// SIMATIC S7-200 SMART project (STEP 7-Micro/WIN SMART), CPU ST30

SYMBOL_TABLE 系统符号
Always_On        SM0.0    // 始终接通
First_Scan_On    SM0.1    // 仅在第一个扫描周期时接通
Time_0_Intrvl    SMB34    // 指定中断 0 的时间间隔（从 5 到 255，以 1 毫秒递增）。
END_SYMBOL_TABLE

ORGANIZATION_BLOCK MAIN:OB1
TITLE=程序注释
BEGIN
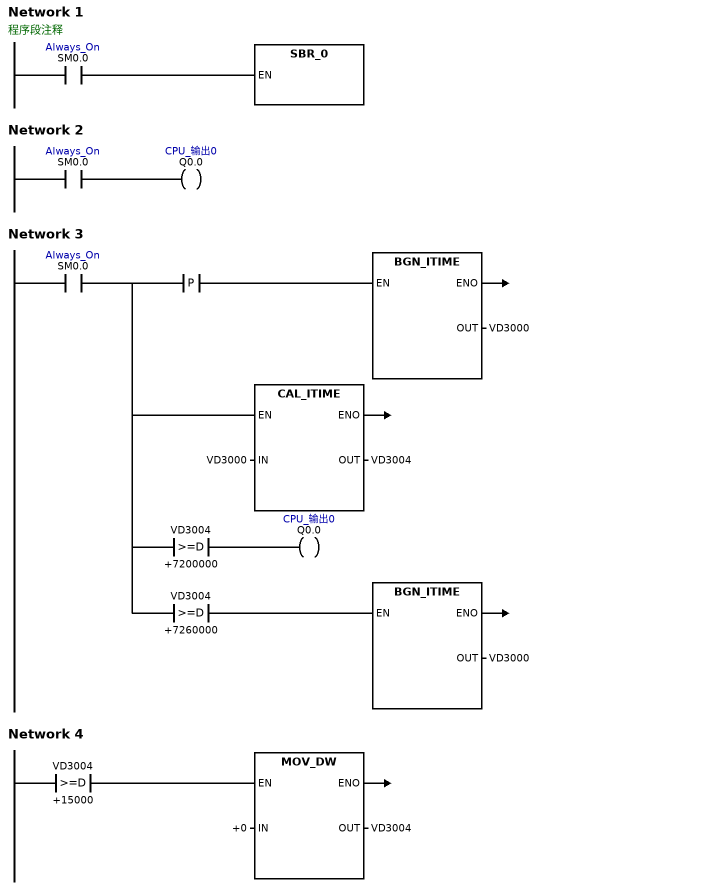
Network 1
// 程序段注释
LD     Always_On:SM0.0
CALL   SBR_0:SBR0
Network 2
LD     Always_On:SM0.0
=      CPU_输出0:Q0.0
Network 3
LD     Always_On:SM0.0
LPS
EU
BITIM  VD3000
LRD
CITIM  VD3000, VD3004
LRD
AD>=   VD3004, +7200000
=      CPU_输出0:Q0.0
LPP
AD>=   VD3004, +7260000
BITIM  VD3000
Network 4
LDD>=  VD3004, +15000
MOVD   +0, VD3004
END_ORGANIZATION_BLOCK

SUBROUTINE_BLOCK SBR_0:SBR0
TITLE=子程序注释
BEGIN
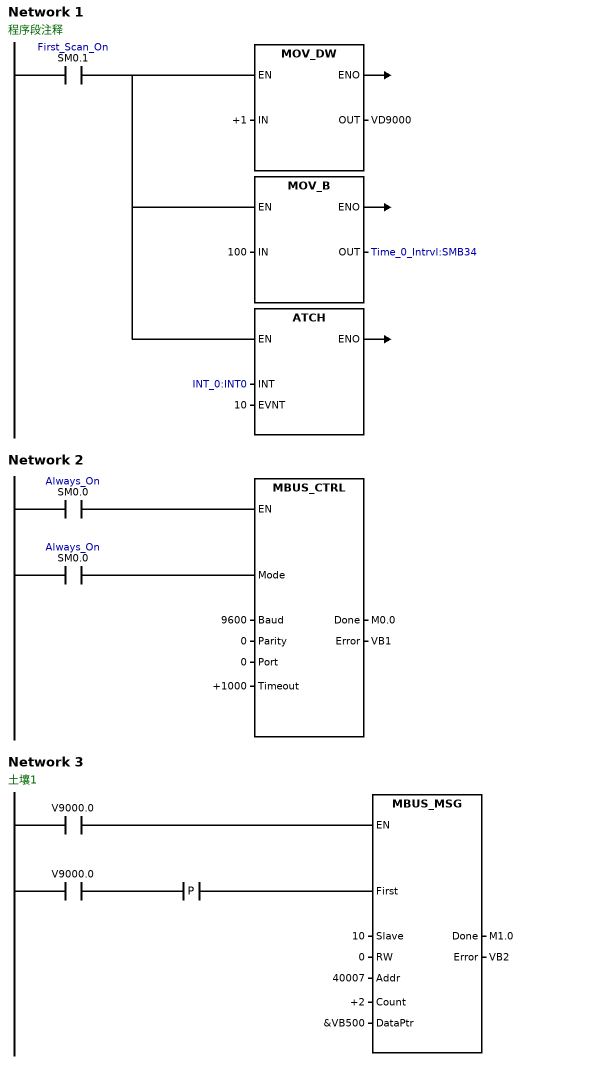
Network 1
// 程序段注释
LD     First_Scan_On:SM0.1
MOVD   +1, VD9000
MOVB   100, Time_0_Intrvl:SMB34
ATCH   INT_0:INT0, 10
Network 2
LD     Always_On:SM0.0
=      L60.0
LD     Always_On:SM0.0
=      L63.7
LD     L60.0
CALL   MBUS_CTRL:SBR1, L63.7, 9600, 0, 0, +1000, M0.0, VB1
Network 3
// 土壤1
LD     V9000.0
=      L60.0
LD     V9000.0
EU
=      L63.7
LD     L60.0
CALL   MBUS_MSG:SBR2, L63.7, 10, 0, 40007, +2, &VB500, M1.0, VB2
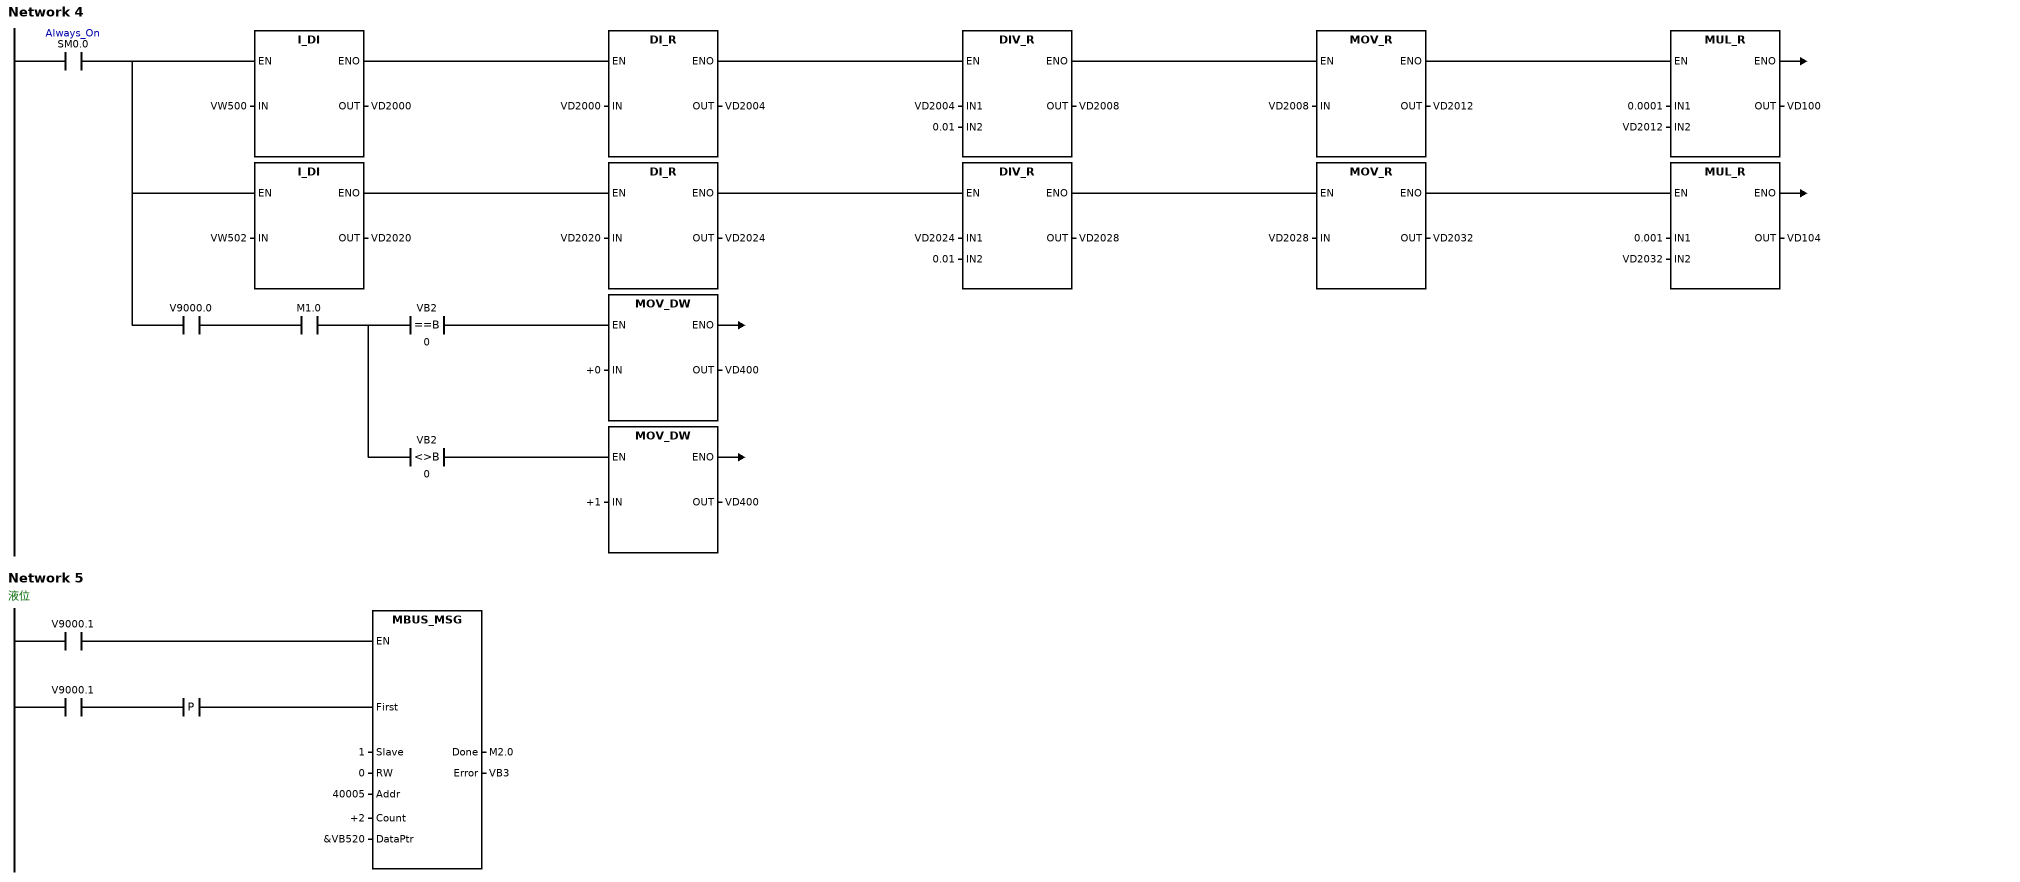
Network 4
LD     Always_On:SM0.0
LPS
ITD    VW500, VD2000
AENO
DTR    VD2000, VD2004
AENO
MOVR   VD2004, VD2008
AENO
/R     0.01, VD2008
AENO
MOVR   VD2008, VD2012
AENO
MOVR   0.0001, VD100
*R     VD2012, VD100
LRD
ITD    VW502, VD2020
AENO
DTR    VD2020, VD2024
AENO
MOVR   VD2024, VD2028
AENO
/R     0.01, VD2028
AENO
MOVR   VD2028, VD2032
AENO
MOVR   0.001, VD104
*R     VD2032, VD104
LPP
A      V9000.0
A      M1.0
LPS
AB=    VB2, 0
MOVD   +0, VD400
LPP
AB<>   VB2, 0
MOVD   +1, VD400
Network 5
// 液位
LD     V9000.1
=      L60.0
LD     V9000.1
EU
=      L63.7
LD     L60.0
CALL   MBUS_MSG:SBR2, L63.7, 1, 0, 40005, +2, &VB520, M2.0, VB3
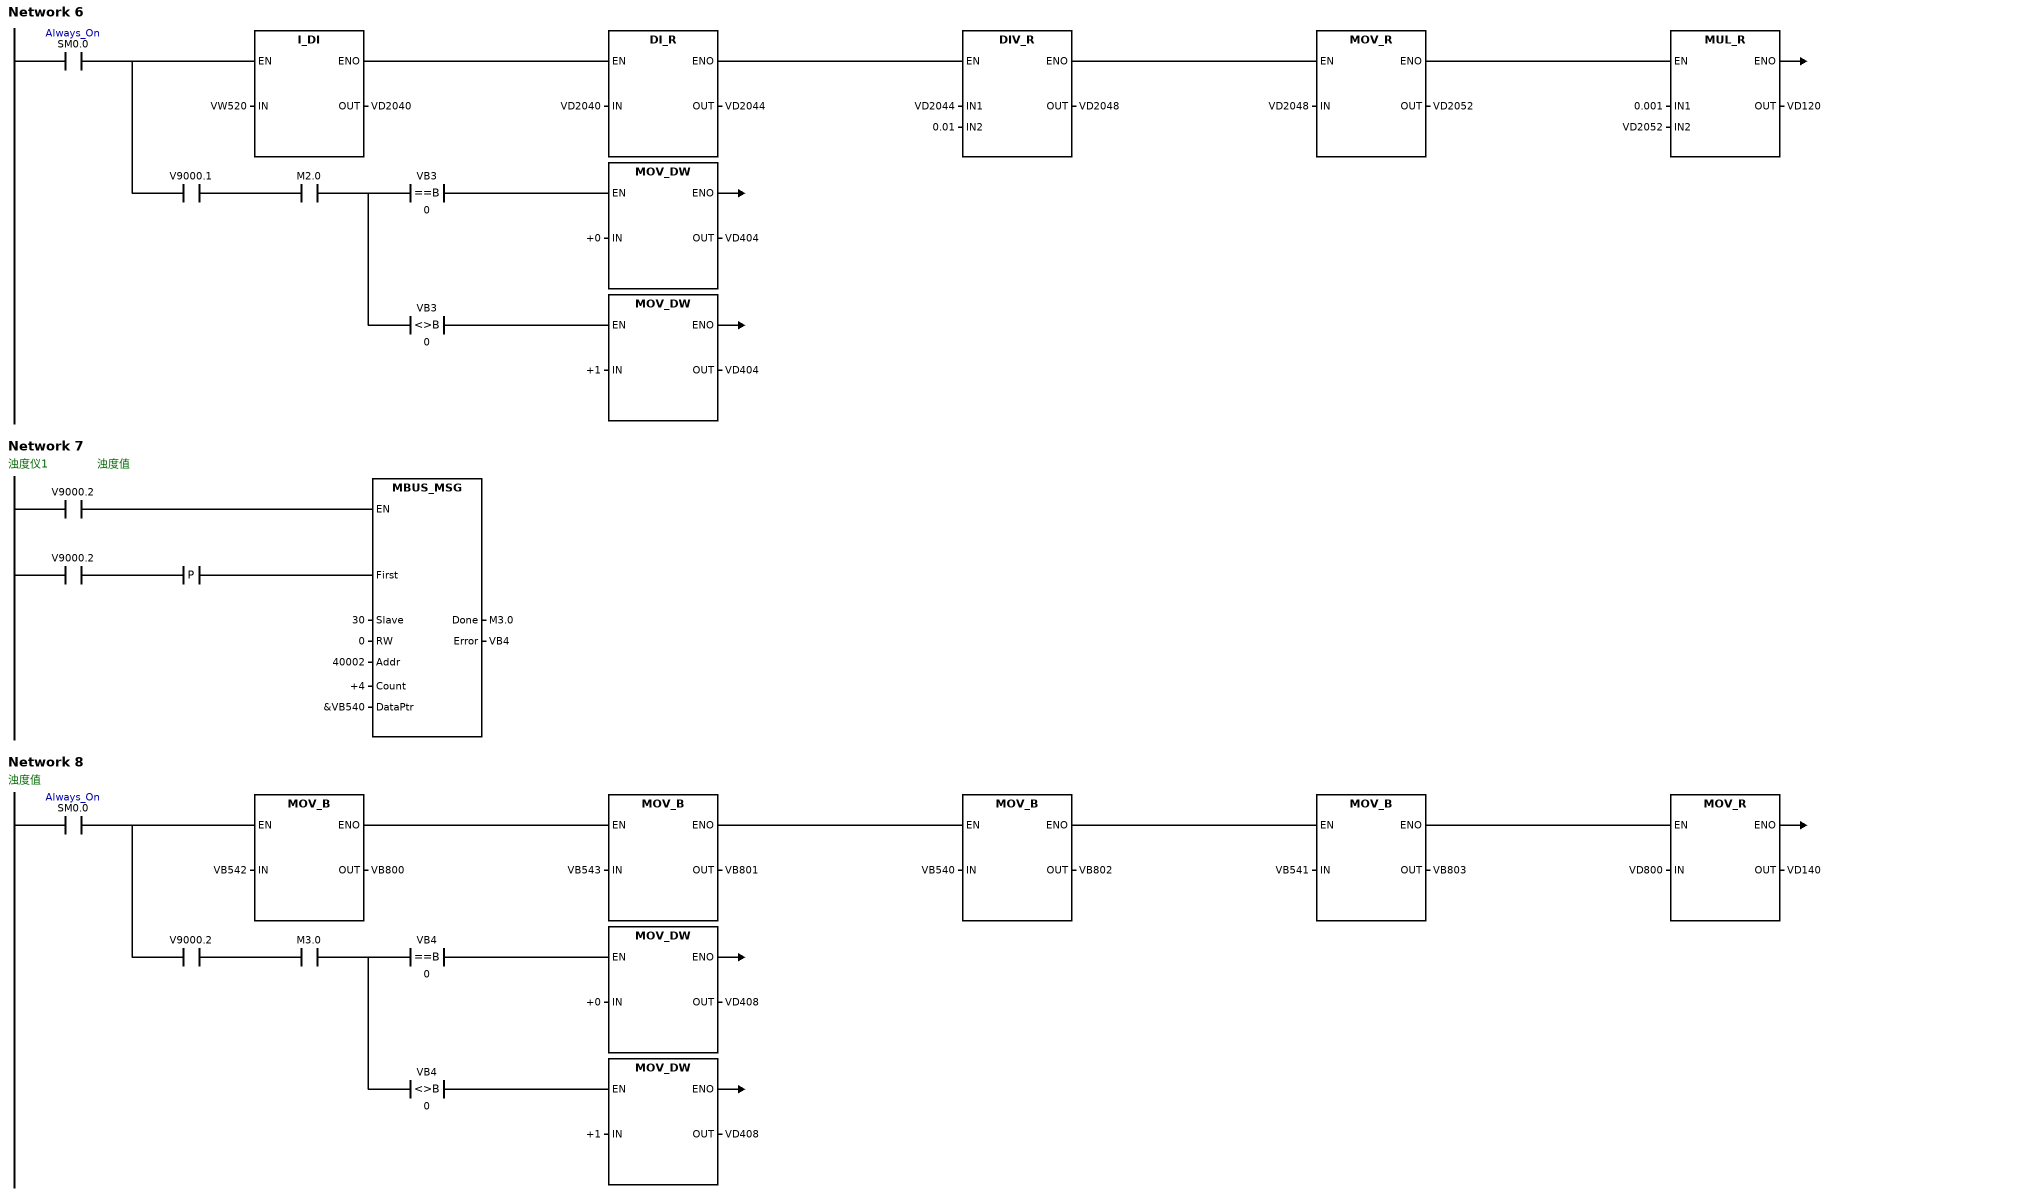
Network 6
LD     Always_On:SM0.0
LPS
ITD    VW520, VD2040
AENO
DTR    VD2040, VD2044
AENO
MOVR   VD2044, VD2048
AENO
/R     0.01, VD2048
AENO
MOVR   VD2048, VD2052
AENO
MOVR   0.001, VD120
*R     VD2052, VD120
LPP
A      V9000.1
A      M2.0
LPS
AB=    VB3, 0
MOVD   +0, VD404
LPP
AB<>   VB3, 0
MOVD   +1, VD404
Network 7
// 浊度仪1              浊度值
LD     V9000.2
=      L60.0
LD     V9000.2
EU
=      L63.7
LD     L60.0
CALL   MBUS_MSG:SBR2, L63.7, 30, 0, 40002, +4, &VB540, M3.0, VB4
Network 8
//  浊度值
LD     Always_On:SM0.0
LPS
MOVB   VB542, VB800
AENO
MOVB   VB543, VB801
AENO
MOVB   VB540, VB802
AENO
MOVB   VB541, VB803
AENO
MOVR   VD800, VD140
LPP
A      V9000.2
A      M3.0
LPS
AB=    VB4, 0
MOVD   +0, VD408
LPP
AB<>   VB4, 0
MOVD   +1, VD408
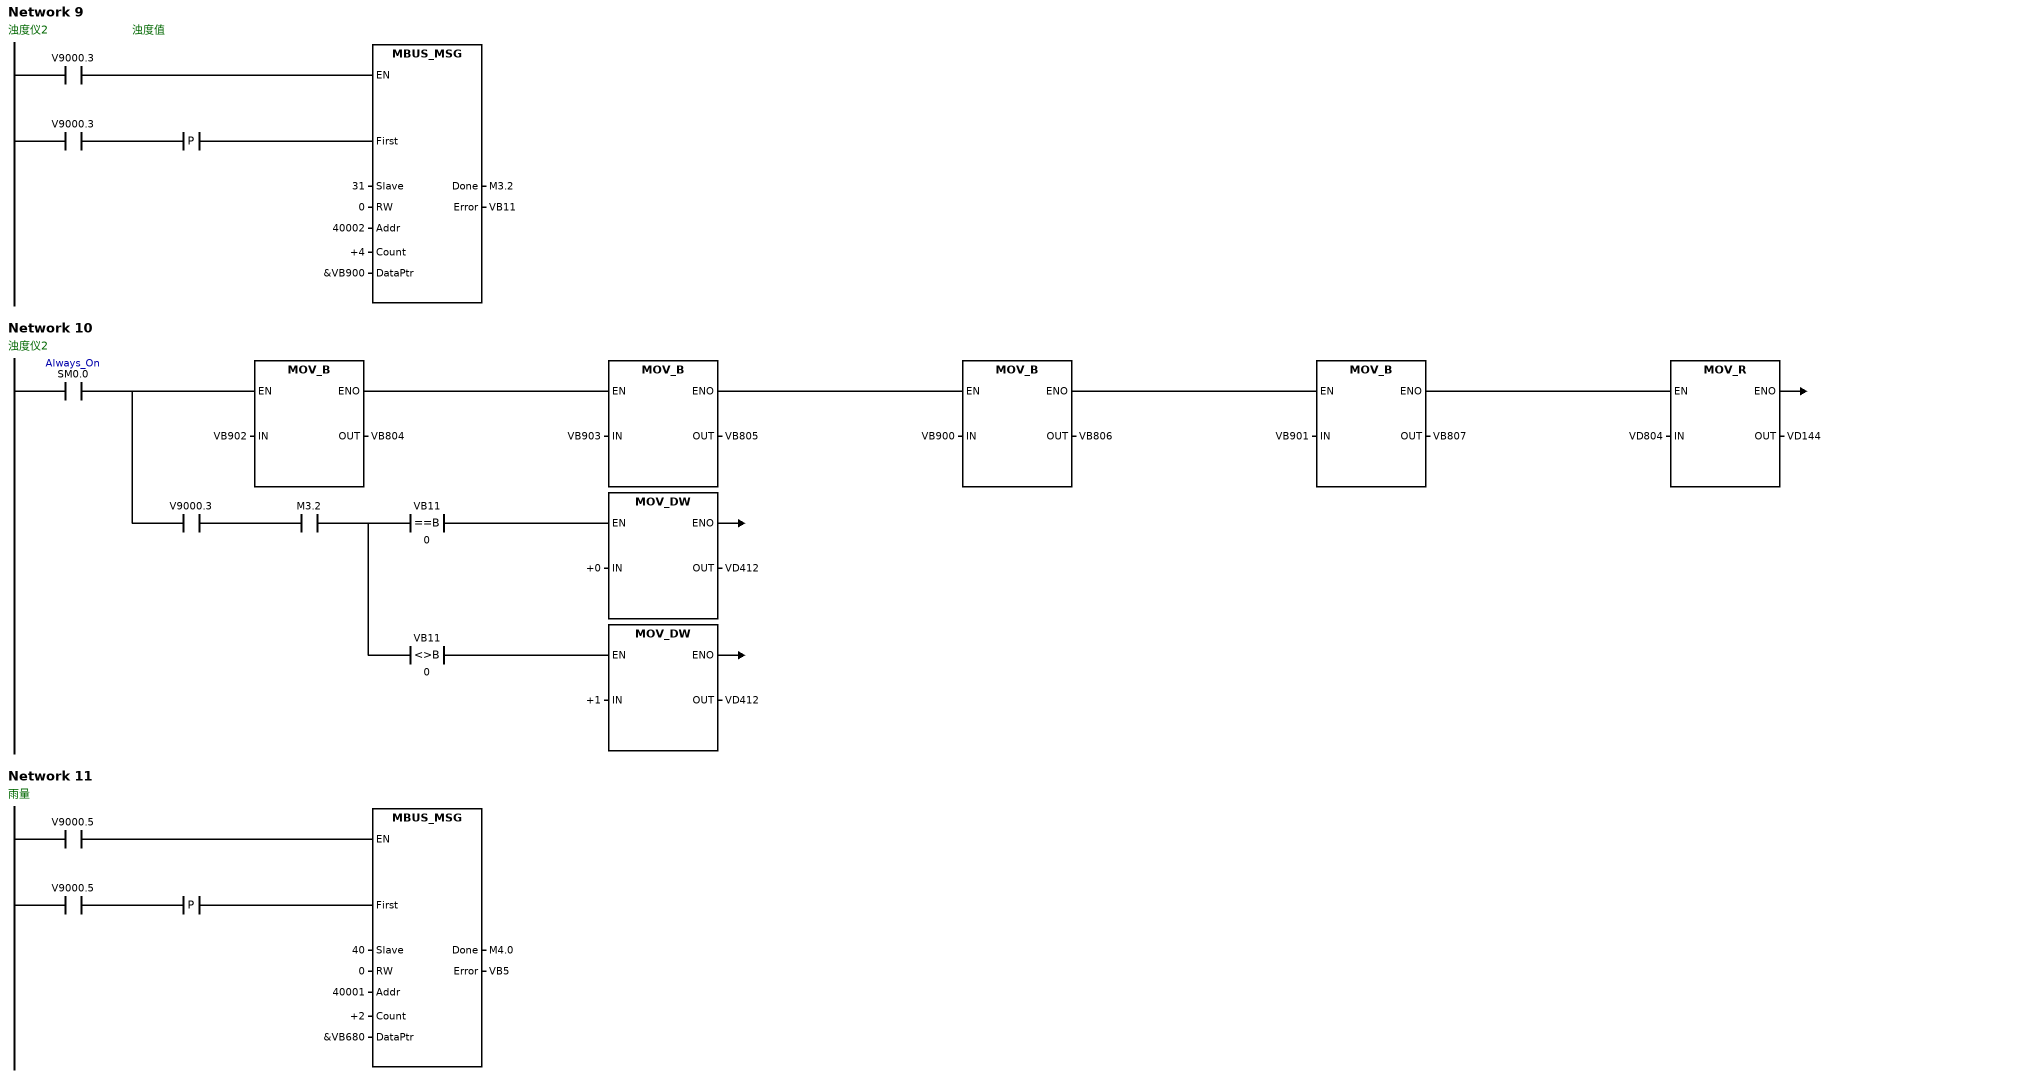
Network 9
// 浊度仪2                        浊度值
LD     V9000.3
=      L60.0
LD     V9000.3
EU
=      L63.7
LD     L60.0
CALL   MBUS_MSG:SBR2, L63.7, 31, 0, 40002, +4, &VB900, M3.2, VB11
Network 10
// 浊度仪2
LD     Always_On:SM0.0
LPS
MOVB   VB902, VB804
AENO
MOVB   VB903, VB805
AENO
MOVB   VB900, VB806
AENO
MOVB   VB901, VB807
AENO
MOVR   VD804, VD144
LPP
A      V9000.3
A      M3.2
LPS
AB=    VB11, 0
MOVD   +0, VD412
LPP
AB<>   VB11, 0
MOVD   +1, VD412
Network 11
// 雨量
LD     V9000.5
=      L60.0
LD     V9000.5
EU
=      L63.7
LD     L60.0
CALL   MBUS_MSG:SBR2, L63.7, 40, 0, 40001, +2, &VB680, M4.0, VB5
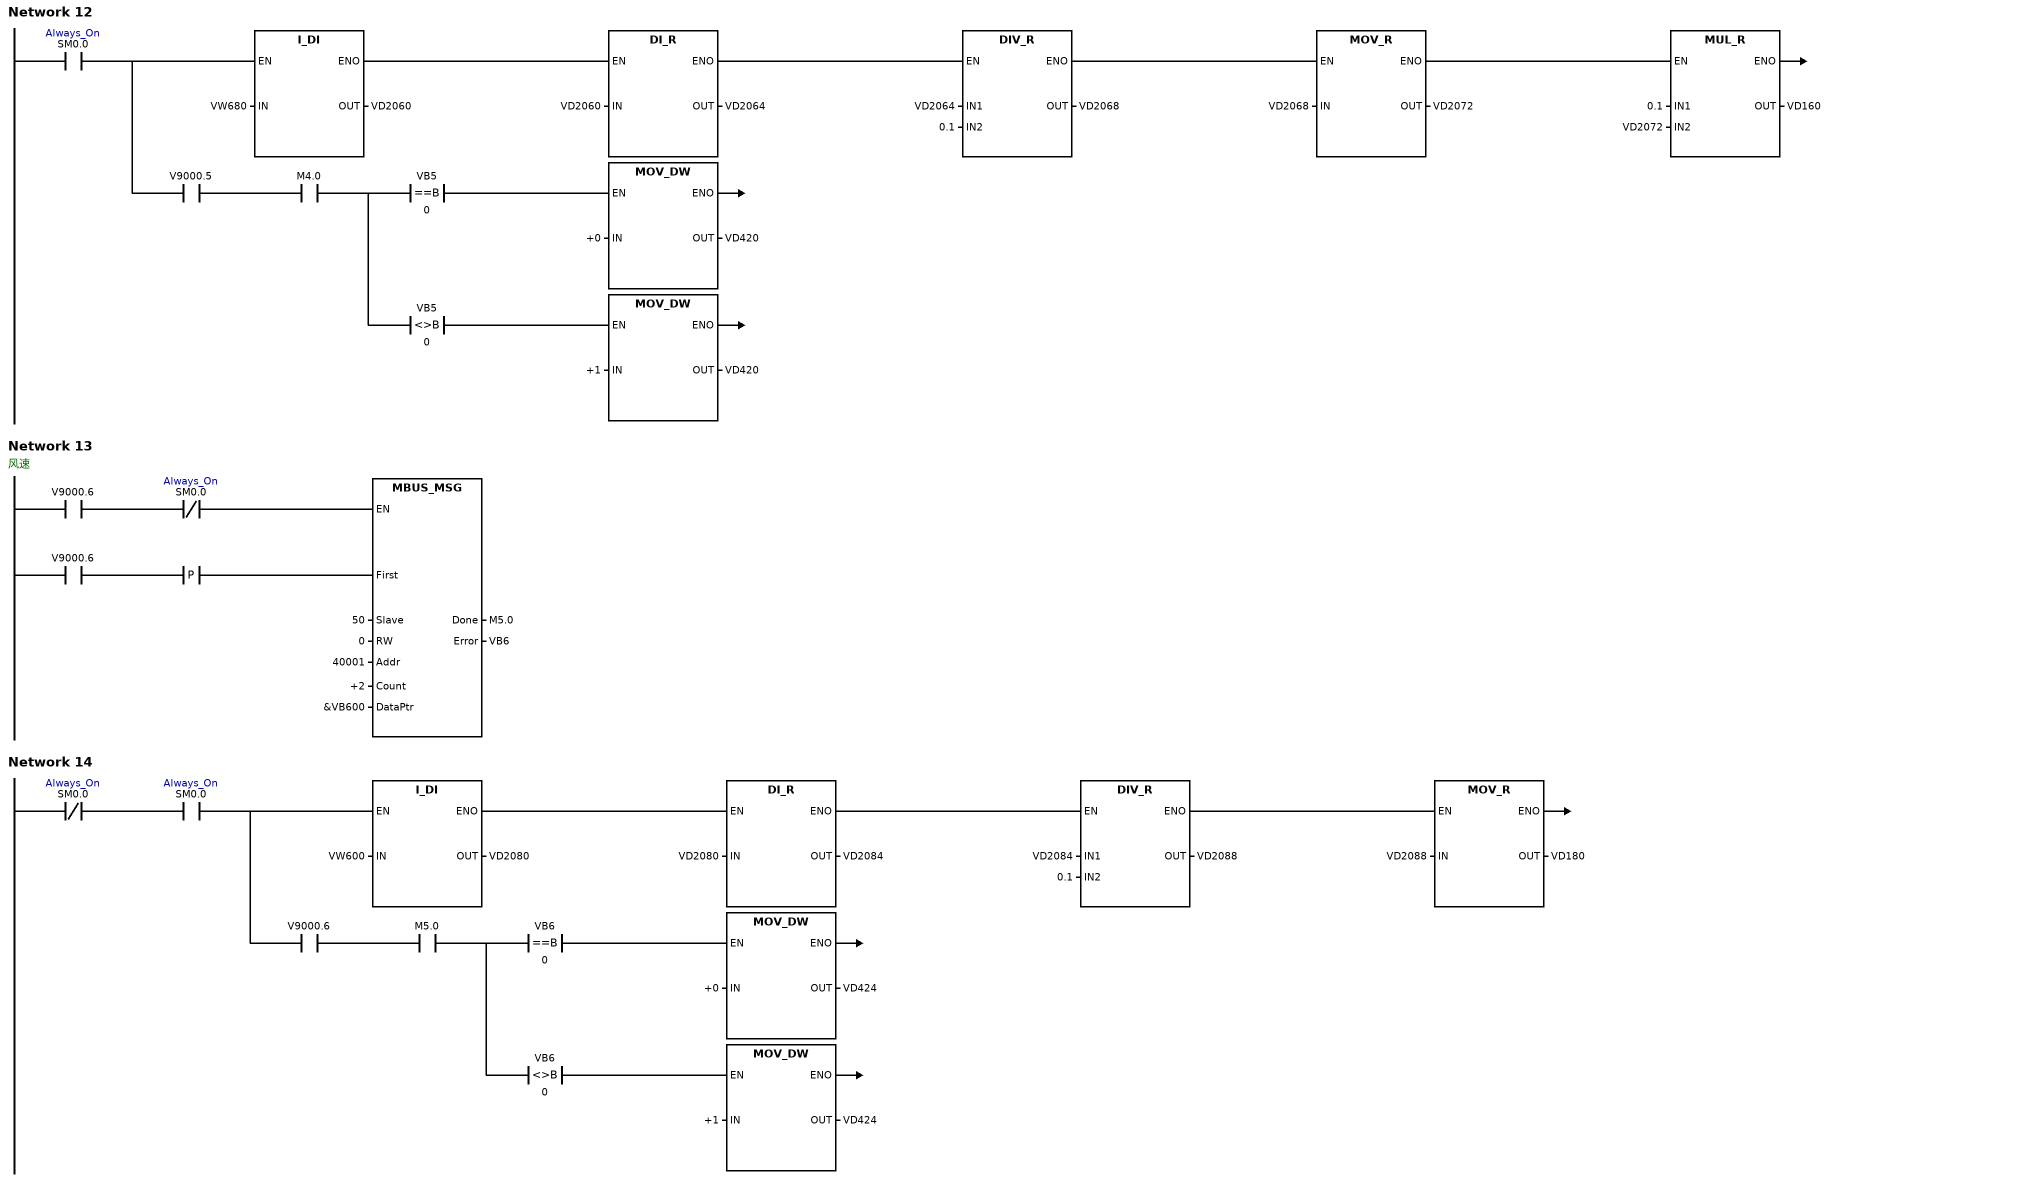
Network 12
LD     Always_On:SM0.0
LPS
ITD    VW680, VD2060
AENO
DTR    VD2060, VD2064
AENO
MOVR   VD2064, VD2068
AENO
/R     0.1, VD2068
AENO
MOVR   VD2068, VD2072
AENO
MOVR   0.1, VD160
*R     VD2072, VD160
LPP
A      V9000.5
A      M4.0
LPS
AB=    VB5, 0
MOVD   +0, VD420
LPP
AB<>   VB5, 0
MOVD   +1, VD420
Network 13
// 风速
LD     V9000.6
AN     Always_On:SM0.0
=      L60.0
LD     V9000.6
EU
=      L63.7
LD     L60.0
CALL   MBUS_MSG:SBR2, L63.7, 50, 0, 40001, +2, &VB600, M5.0, VB6
Network 14
LDN    Always_On:SM0.0
A      Always_On:SM0.0
LPS
ITD    VW600, VD2080
AENO
DTR    VD2080, VD2084
AENO
MOVR   VD2084, VD2088
AENO
/R     0.1, VD2088
AENO
MOVR   VD2088, VD180
LPP
A      V9000.6
A      M5.0
LPS
AB=    VB6, 0
MOVD   +0, VD424
LPP
AB<>   VB6, 0
MOVD   +1, VD424
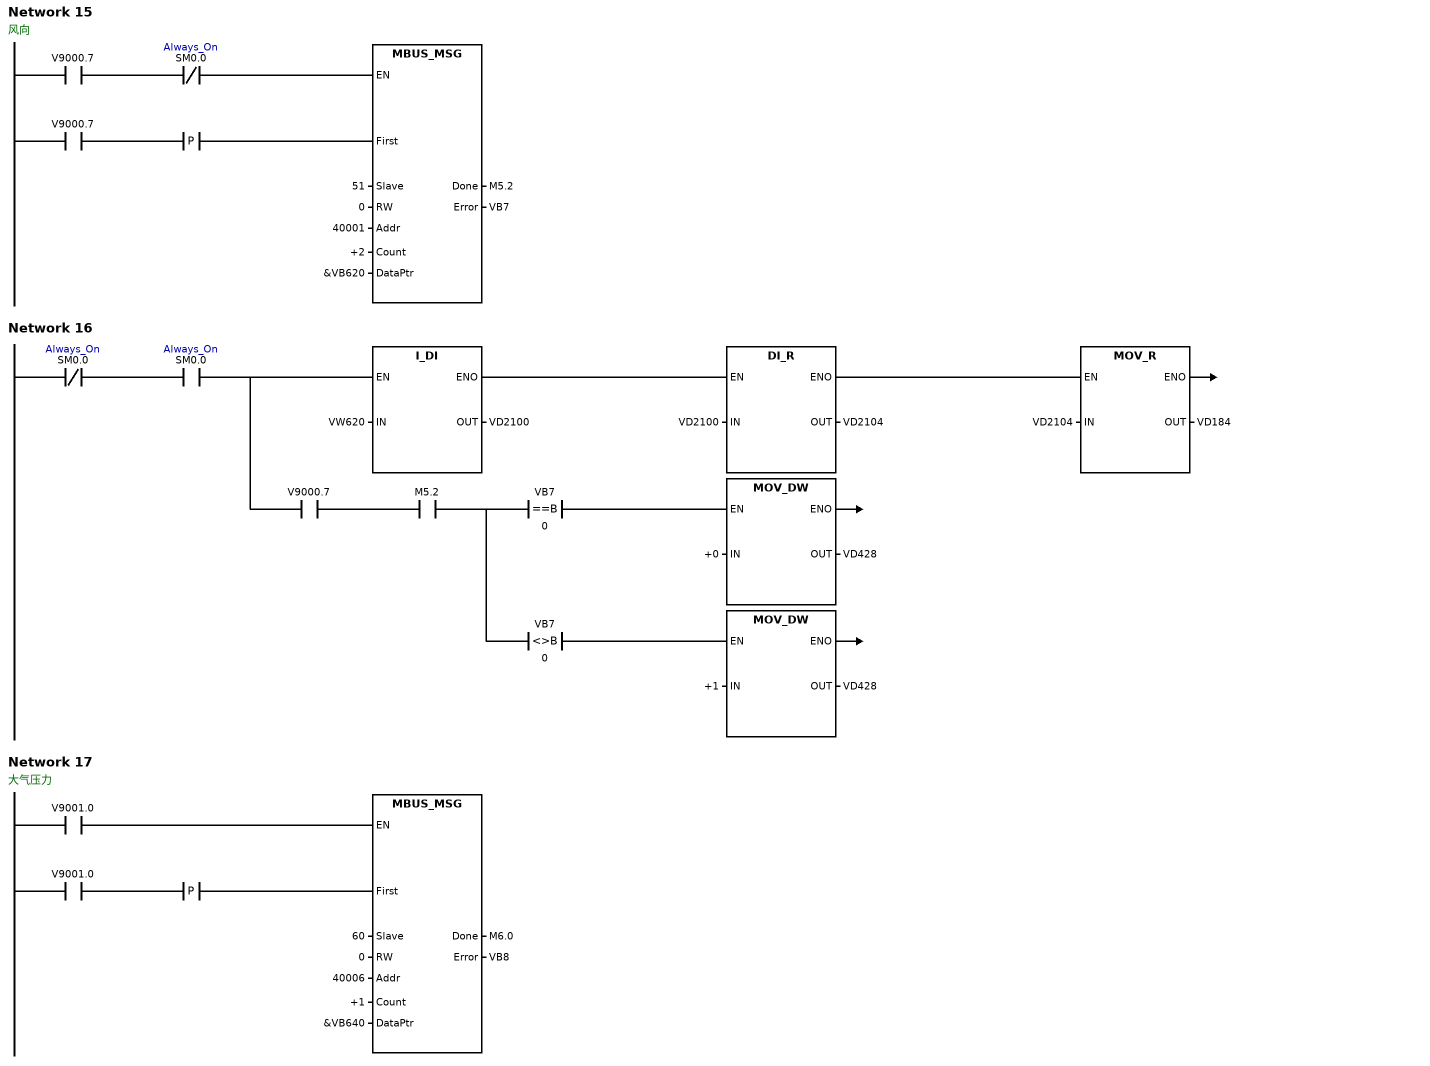
Network 15
// 风向
LD     V9000.7
AN     Always_On:SM0.0
=      L60.0
LD     V9000.7
EU
=      L63.7
LD     L60.0
CALL   MBUS_MSG:SBR2, L63.7, 51, 0, 40001, +2, &VB620, M5.2, VB7
Network 16
LDN    Always_On:SM0.0
A      Always_On:SM0.0
LPS
ITD    VW620, VD2100
AENO
DTR    VD2100, VD2104
AENO
MOVR   VD2104, VD184
LPP
A      V9000.7
A      M5.2
LPS
AB=    VB7, 0
MOVD   +0, VD428
LPP
AB<>   VB7, 0
MOVD   +1, VD428
Network 17
// 大气压力
LD     V9001.0
=      L60.0
LD     V9001.0
EU
=      L63.7
LD     L60.0
CALL   MBUS_MSG:SBR2, L63.7, 60, 0, 40006, +1, &VB640, M6.0, VB8
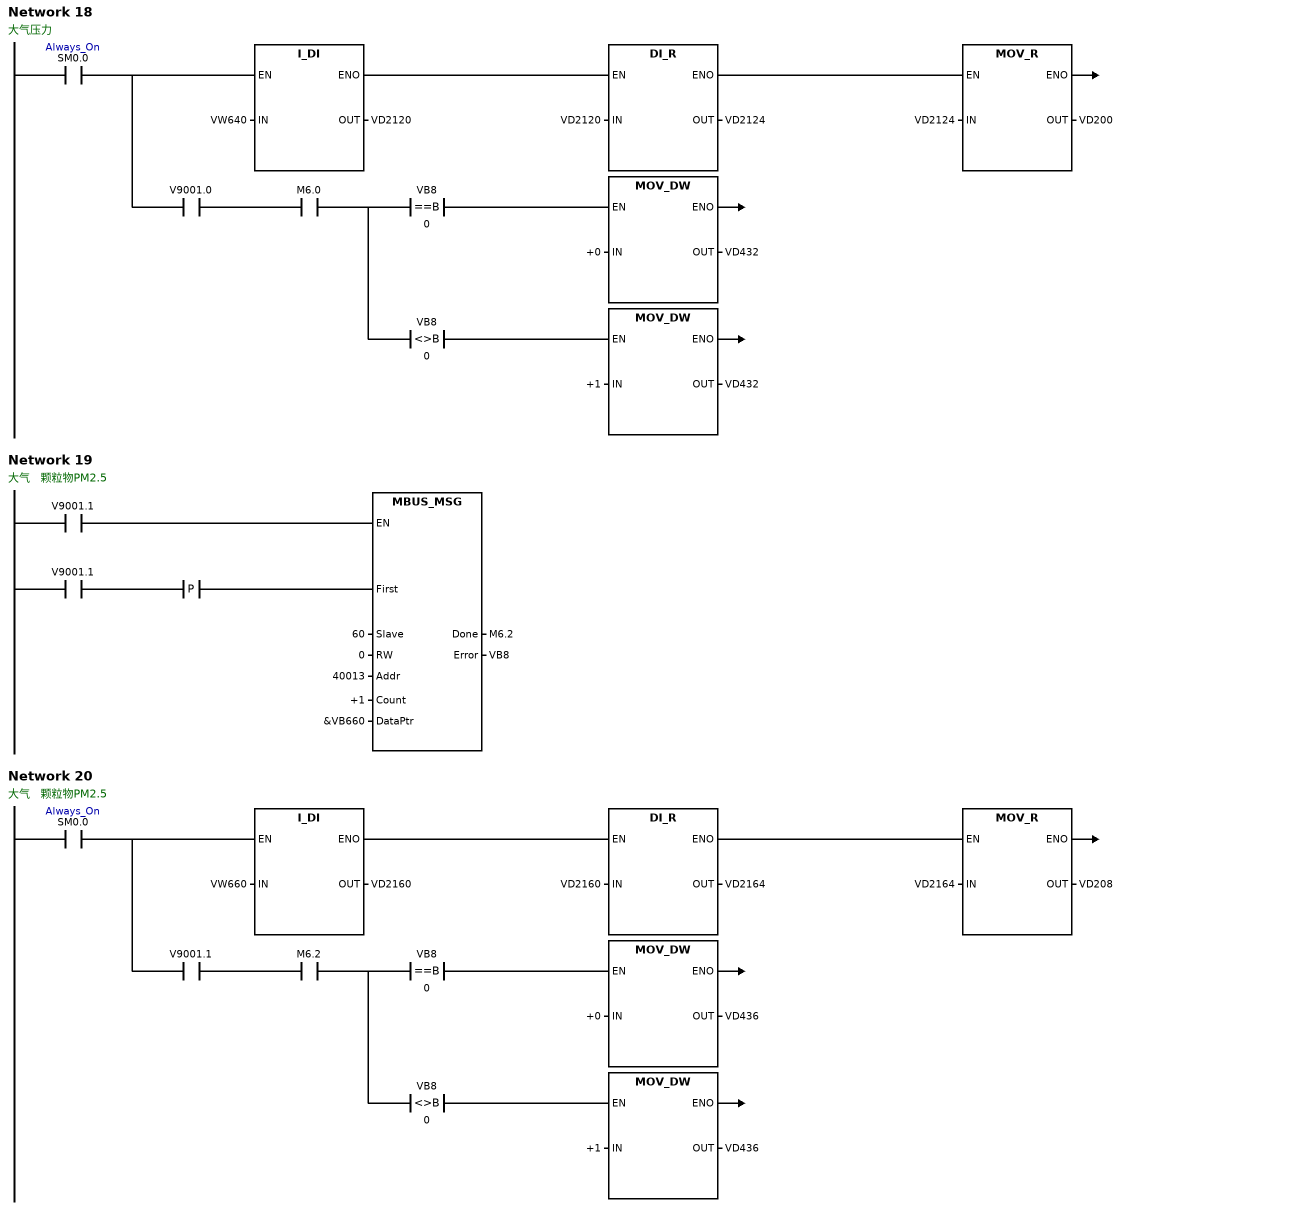
Network 18
// 大气压力
LD     Always_On:SM0.0
LPS
ITD    VW640, VD2120
AENO
DTR    VD2120, VD2124
AENO
MOVR   VD2124, VD200
LPP
A      V9001.0
A      M6.0
LPS
AB=    VB8, 0
MOVD   +0, VD432
LPP
AB<>   VB8, 0
MOVD   +1, VD432
Network 19
// 大气   颗粒物PM2.5
LD     V9001.1
=      L60.0
LD     V9001.1
EU
=      L63.7
LD     L60.0
CALL   MBUS_MSG:SBR2, L63.7, 60, 0, 40013, +1, &VB660, M6.2, VB8
Network 20
// 大气   颗粒物PM2.5
LD     Always_On:SM0.0
LPS
ITD    VW660, VD2160
AENO
DTR    VD2160, VD2164
AENO
MOVR   VD2164, VD208
LPP
A      V9001.1
A      M6.2
LPS
AB=    VB8, 0
MOVD   +0, VD436
LPP
AB<>   VB8, 0
MOVD   +1, VD436
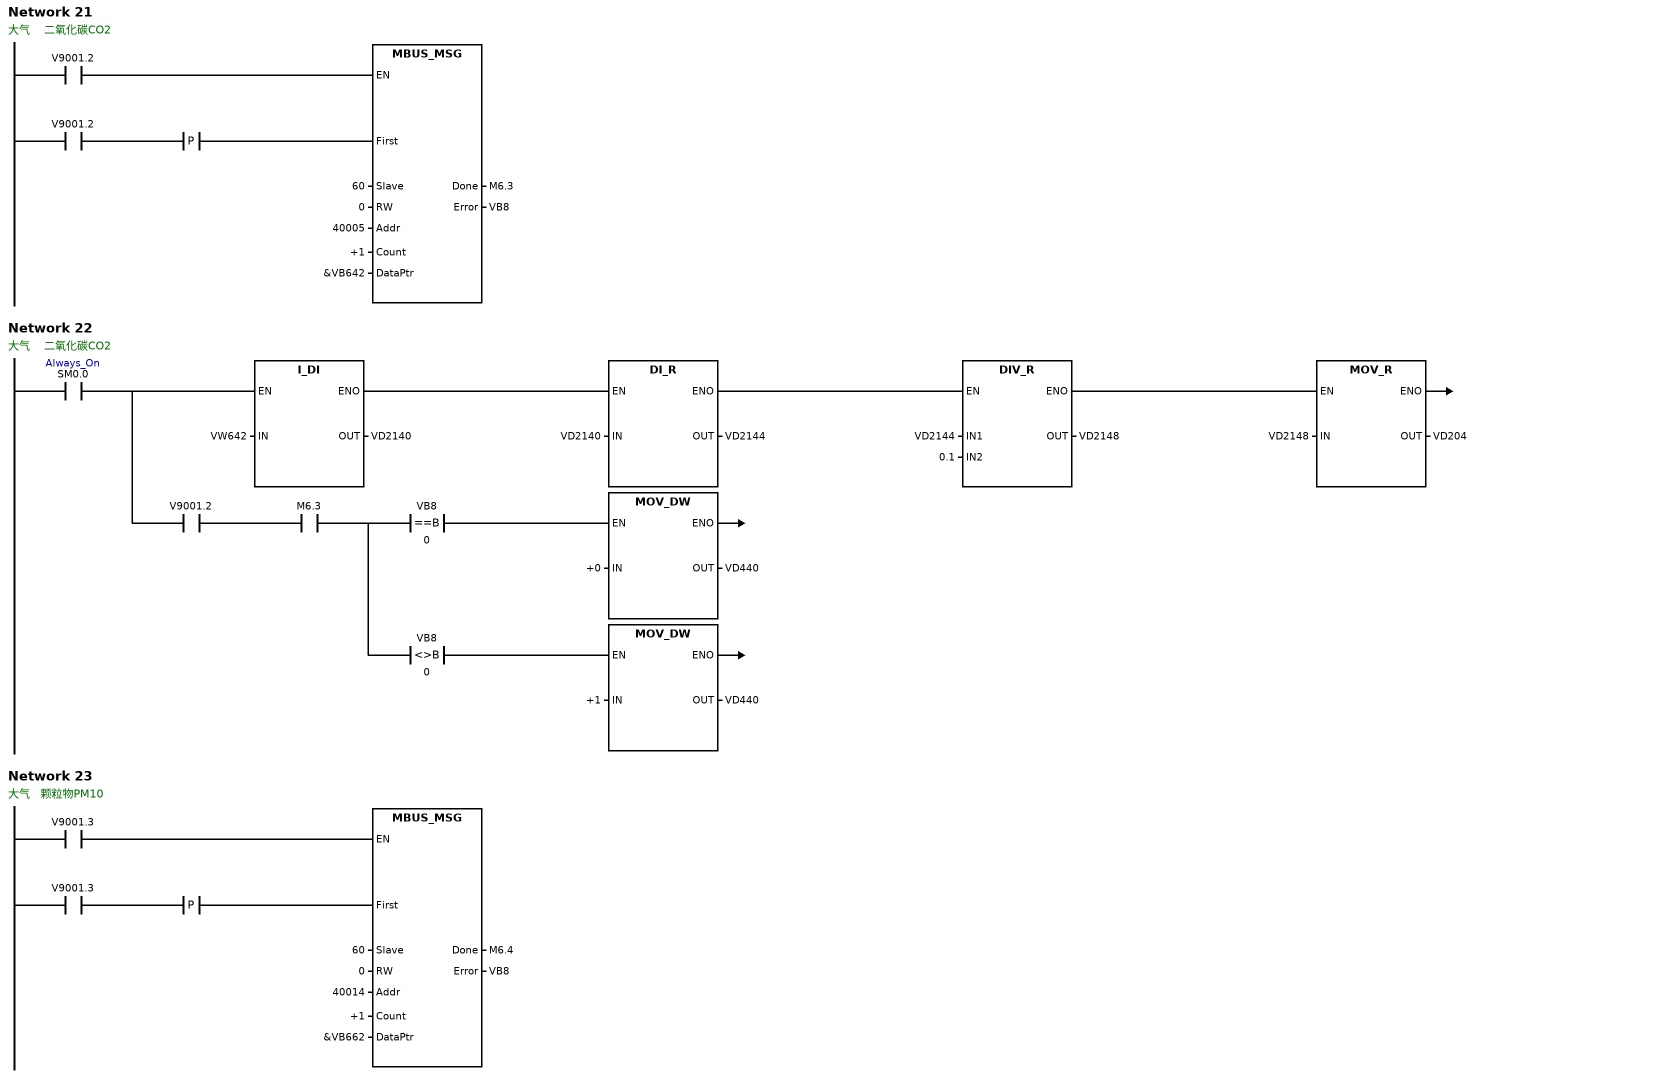
Network 21
// 大气    二氧化碳CO2
LD     V9001.2
=      L60.0
LD     V9001.2
EU
=      L63.7
LD     L60.0
CALL   MBUS_MSG:SBR2, L63.7, 60, 0, 40005, +1, &VB642, M6.3, VB8
Network 22
// 大气    二氧化碳CO2
LD     Always_On:SM0.0
LPS
ITD    VW642, VD2140
AENO
DTR    VD2140, VD2144
AENO
MOVR   VD2144, VD2148
AENO
/R     0.1, VD2148
AENO
MOVR   VD2148, VD204
LPP
A      V9001.2
A      M6.3
LPS
AB=    VB8, 0
MOVD   +0, VD440
LPP
AB<>   VB8, 0
MOVD   +1, VD440
Network 23
// 大气   颗粒物PM10
LD     V9001.3
=      L60.0
LD     V9001.3
EU
=      L63.7
LD     L60.0
CALL   MBUS_MSG:SBR2, L63.7, 60, 0, 40014, +1, &VB662, M6.4, VB8
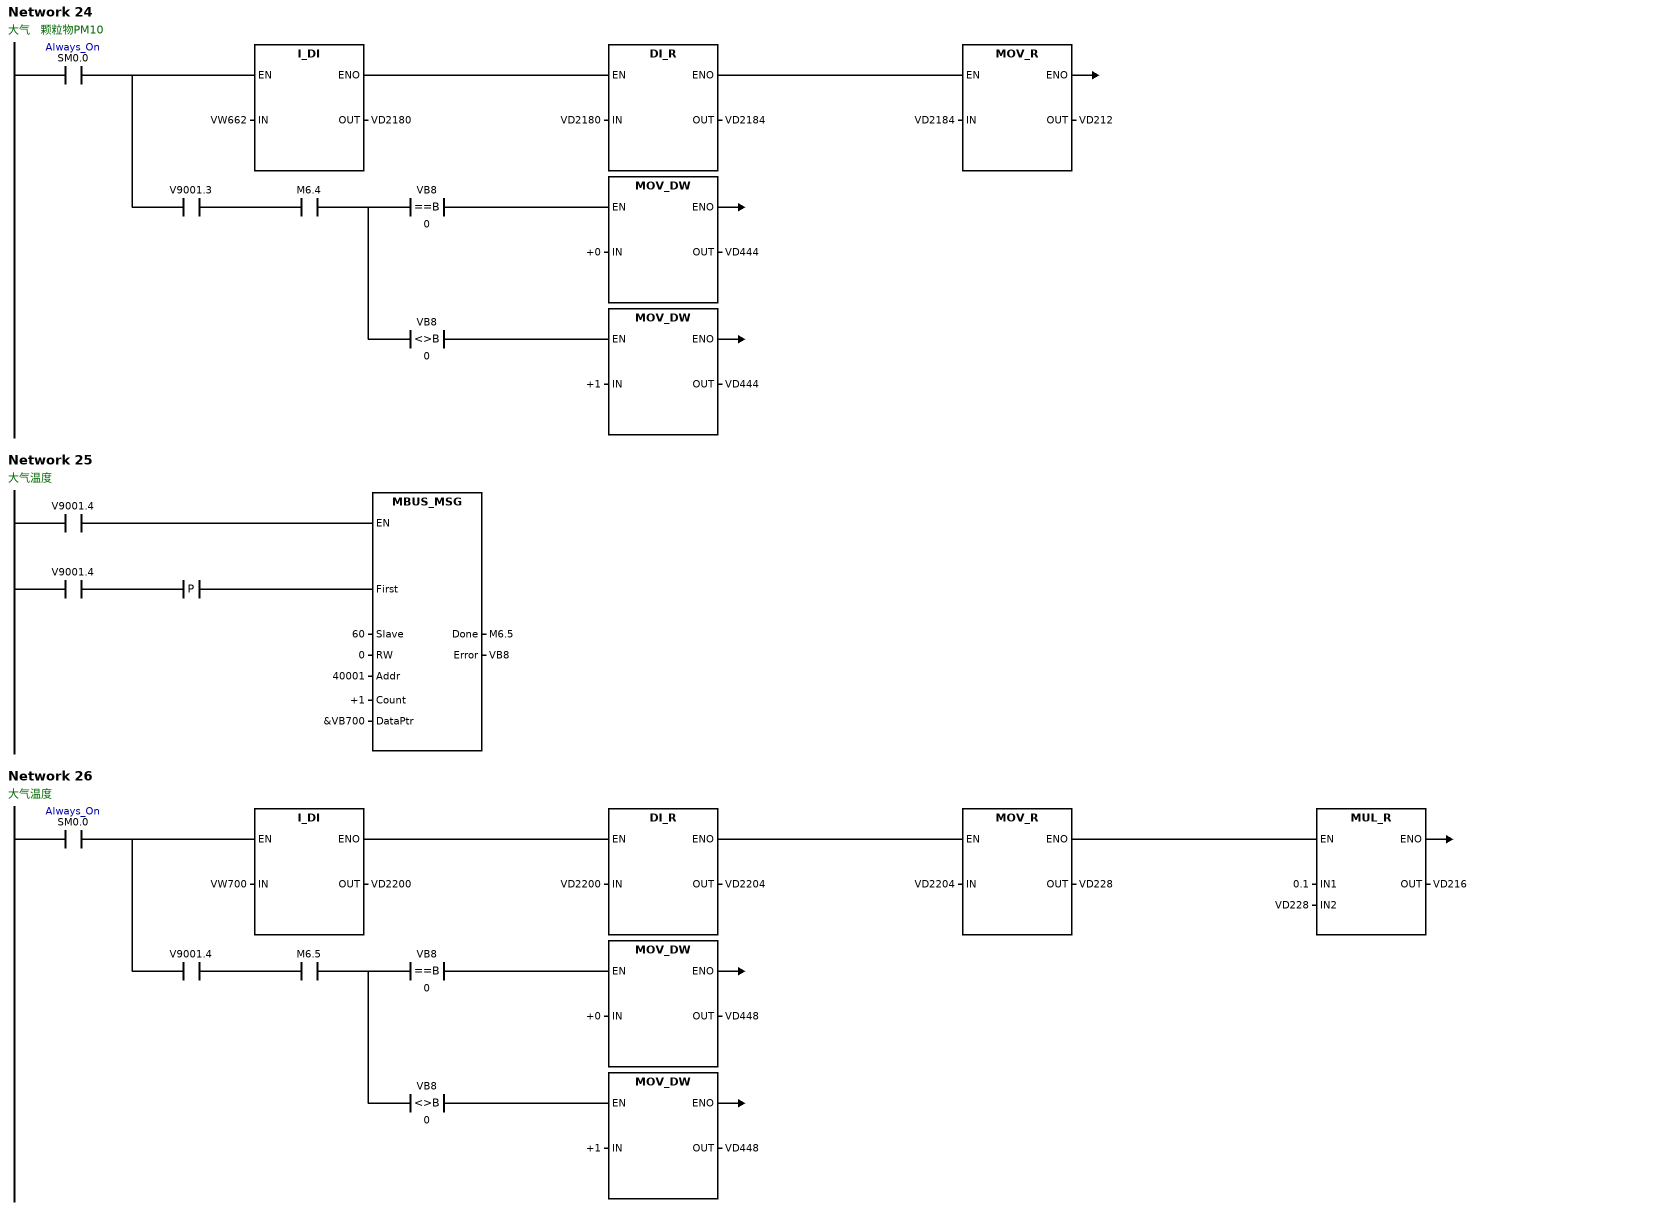
Network 24
// 大气   颗粒物PM10
LD     Always_On:SM0.0
LPS
ITD    VW662, VD2180
AENO
DTR    VD2180, VD2184
AENO
MOVR   VD2184, VD212
LPP
A      V9001.3
A      M6.4
LPS
AB=    VB8, 0
MOVD   +0, VD444
LPP
AB<>   VB8, 0
MOVD   +1, VD444
Network 25
// 大气温度
LD     V9001.4
=      L60.0
LD     V9001.4
EU
=      L63.7
LD     L60.0
CALL   MBUS_MSG:SBR2, L63.7, 60, 0, 40001, +1, &VB700, M6.5, VB8
Network 26
// 大气温度
LD     Always_On:SM0.0
LPS
ITD    VW700, VD2200
AENO
DTR    VD2200, VD2204
AENO
MOVR   VD2204, VD228
AENO
MOVR   0.1, VD216
*R     VD228, VD216
LPP
A      V9001.4
A      M6.5
LPS
AB=    VB8, 0
MOVD   +0, VD448
LPP
AB<>   VB8, 0
MOVD   +1, VD448
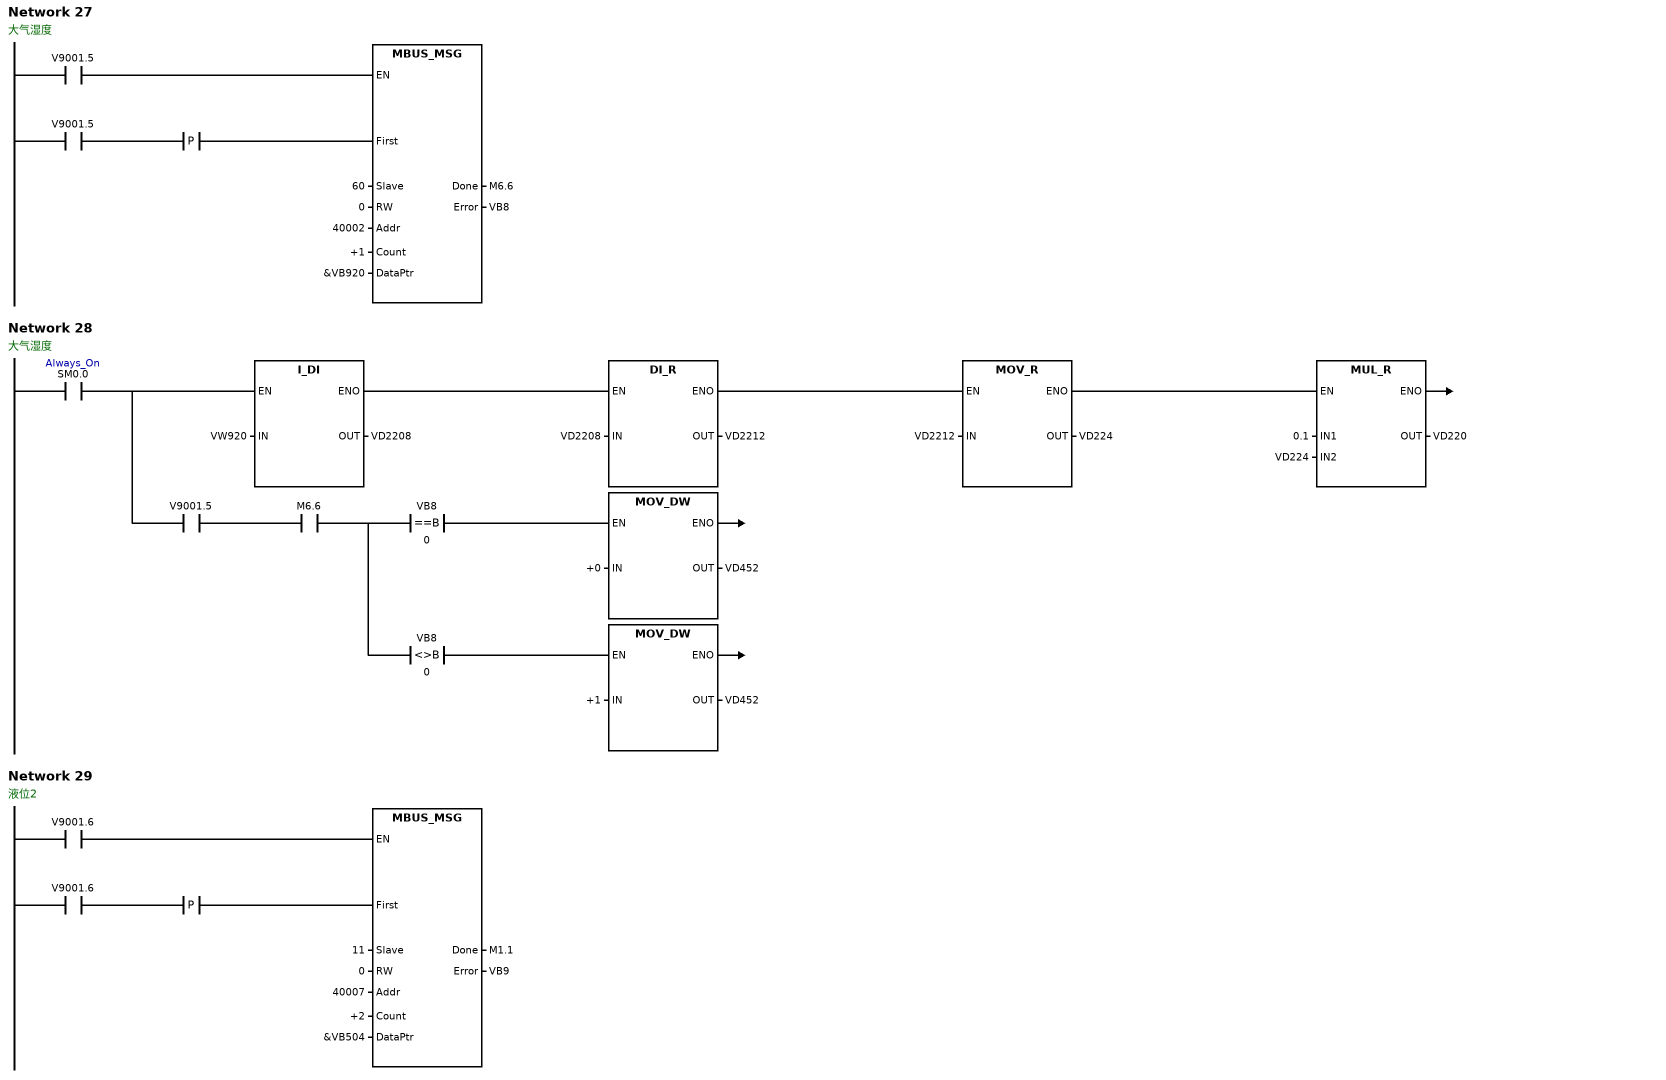
Network 27
// 大气湿度
LD     V9001.5
=      L60.0
LD     V9001.5
EU
=      L63.7
LD     L60.0
CALL   MBUS_MSG:SBR2, L63.7, 60, 0, 40002, +1, &VB920, M6.6, VB8
Network 28
// 大气湿度
LD     Always_On:SM0.0
LPS
ITD    VW920, VD2208
AENO
DTR    VD2208, VD2212
AENO
MOVR   VD2212, VD224
AENO
MOVR   0.1, VD220
*R     VD224, VD220
LPP
A      V9001.5
A      M6.6
LPS
AB=    VB8, 0
MOVD   +0, VD452
LPP
AB<>   VB8, 0
MOVD   +1, VD452
Network 29
// 液位2
LD     V9001.6
=      L60.0
LD     V9001.6
EU
=      L63.7
LD     L60.0
CALL   MBUS_MSG:SBR2, L63.7, 11, 0, 40007, +2, &VB504, M1.1, VB9
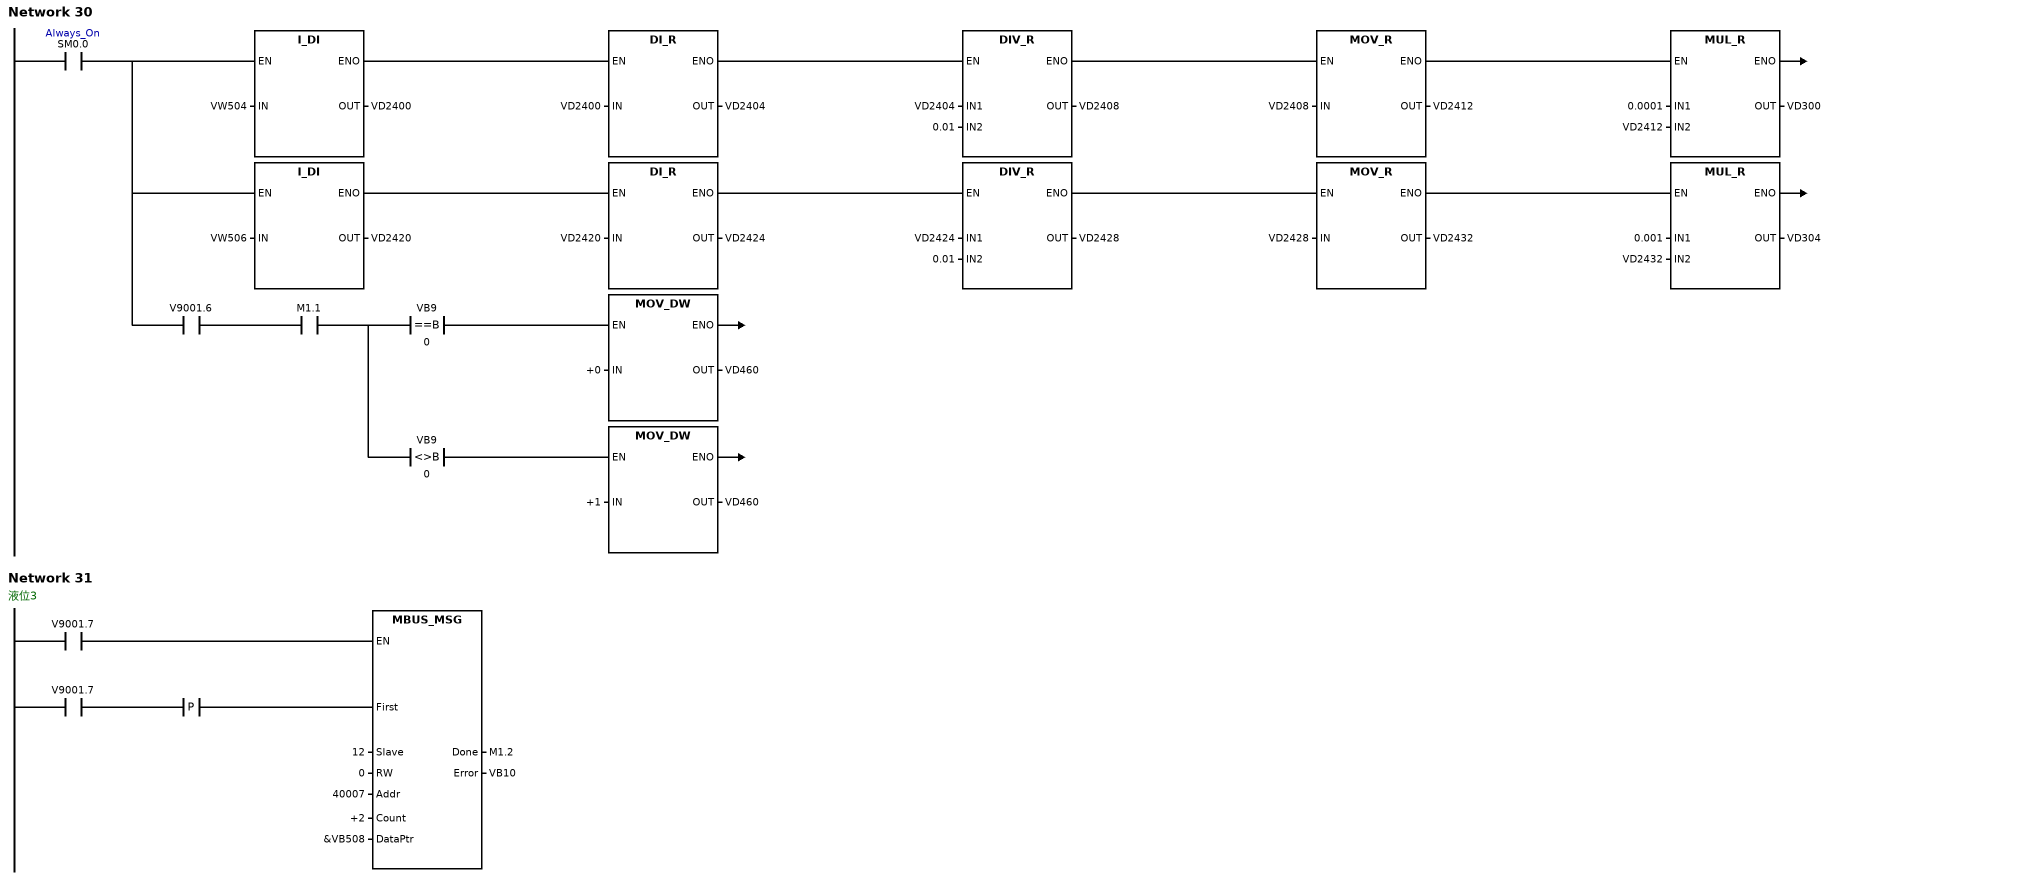
Network 30
LD     Always_On:SM0.0
LPS
ITD    VW504, VD2400
AENO
DTR    VD2400, VD2404
AENO
MOVR   VD2404, VD2408
AENO
/R     0.01, VD2408
AENO
MOVR   VD2408, VD2412
AENO
MOVR   0.0001, VD300
*R     VD2412, VD300
LRD
ITD    VW506, VD2420
AENO
DTR    VD2420, VD2424
AENO
MOVR   VD2424, VD2428
AENO
/R     0.01, VD2428
AENO
MOVR   VD2428, VD2432
AENO
MOVR   0.001, VD304
*R     VD2432, VD304
LPP
A      V9001.6
A      M1.1
LPS
AB=    VB9, 0
MOVD   +0, VD460
LPP
AB<>   VB9, 0
MOVD   +1, VD460
Network 31
// 液位3
LD     V9001.7
=      L60.0
LD     V9001.7
EU
=      L63.7
LD     L60.0
CALL   MBUS_MSG:SBR2, L63.7, 12, 0, 40007, +2, &VB508, M1.2, VB10
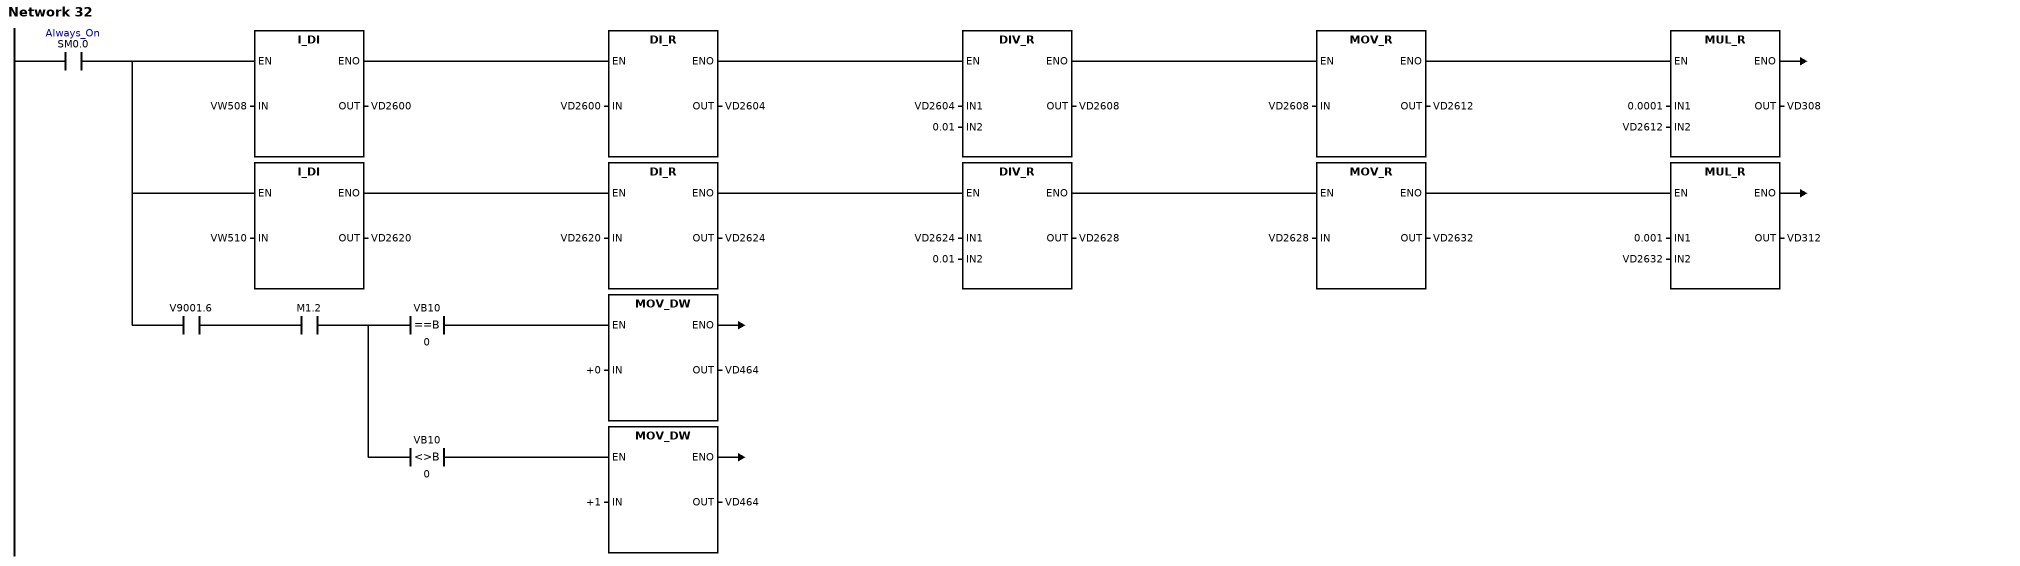
Network 32
LD     Always_On:SM0.0
LPS
ITD    VW508, VD2600
AENO
DTR    VD2600, VD2604
AENO
MOVR   VD2604, VD2608
AENO
/R     0.01, VD2608
AENO
MOVR   VD2608, VD2612
AENO
MOVR   0.0001, VD308
*R     VD2612, VD308
LRD
ITD    VW510, VD2620
AENO
DTR    VD2620, VD2624
AENO
MOVR   VD2624, VD2628
AENO
/R     0.01, VD2628
AENO
MOVR   VD2628, VD2632
AENO
MOVR   0.001, VD312
*R     VD2632, VD312
LPP
A      V9001.6
A      M1.2
LPS
AB=    VB10, 0
MOVD   +0, VD464
LPP
AB<>   VB10, 0
MOVD   +1, VD464
END_SUBROUTINE_BLOCK

// SBR1: protected block, not included

// SBR2: protected block, not included

// SBR3: protected block, not included

INTERRUPT_BLOCK INT_0:INT0
TITLE=中断例程注释
BEGIN
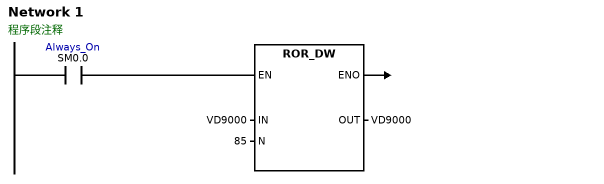
Network 1
// 程序段注释
LD     Always_On:SM0.0
RRD    VD9000, 85
END_INTERRUPT_BLOCK

// INT1: protected block, not included
